TYPE ST_InventerUD EXTENDS ST_Inventer :
STRUCT
	iLowPos			AT %I*:BOOL;		//前往低點位 
	iHighPos		AT %I*:BOOL;		//前往高點位 
END_STRUCT
END_TYPE

(* stored: Version 1.1.0.1, ProductVersion 3.1.4024.15
   DUT ST_InventerUD: Id {d9be18f4-3452-4cd1-89fe-85e6427eae57} *)
